// TIA Portal V19 export
FUNCTION_BLOCK "LineStates"   // FB8, LAD
{ S7_Optimized_Access := 'TRUE' }
// stored: MemoryReserve 100, SetENOAutomatically false
   VAR
      StateM1LineRunning { S7_SetPoint := 'True'} : "GenericState";
      StateM2LineRunning { S7_SetPoint := 'True'} : "GenericState";
      StateM1CurrentOrderNo { S7_SetPoint := 'True'} : "GenericState";
      StateM2CurrentOrderNo { S7_SetPoint := 'True'} : "GenericState";
      PubJsonMqttInstM1LineRunning { S7_SetPoint := 'True'} : "PublishJsonMqtt";
      PubJsonMqttInstM2LineRunning { S7_SetPoint := 'True'} : "PublishJsonMqtt";
      PubJsonMqttInstM1CurrentOrderNo { S7_SetPoint := 'True'} : "PublishJsonMqtt";
      PubJsonMqttInstM2CurrentOrderNo { S7_SetPoint := 'True'} : "PublishJsonMqtt";
      tpGen01 { S7_SetPoint := 'True'} : TP_TIME;
      tpGen02 { S7_SetPoint := 'True'} : TP_TIME;
   END_VAR
   VAR_TEMP   // added for the SCL form of the ladder/FBD networks
      _w1 : Bool;
   END_VAR
BEGIN

REGION Network 1 (SCL): Generator for data publish
   #tpGen01(IN:=NOT #tpGen02.Q,
            PT:=T#4S);

   #tpGen02(IN:=NOT #tpGen01.Q,
            PT:=T#100MS);
END_REGION

REGION Network 2: Line 1 / Machine 1 / State 'LineRunning'
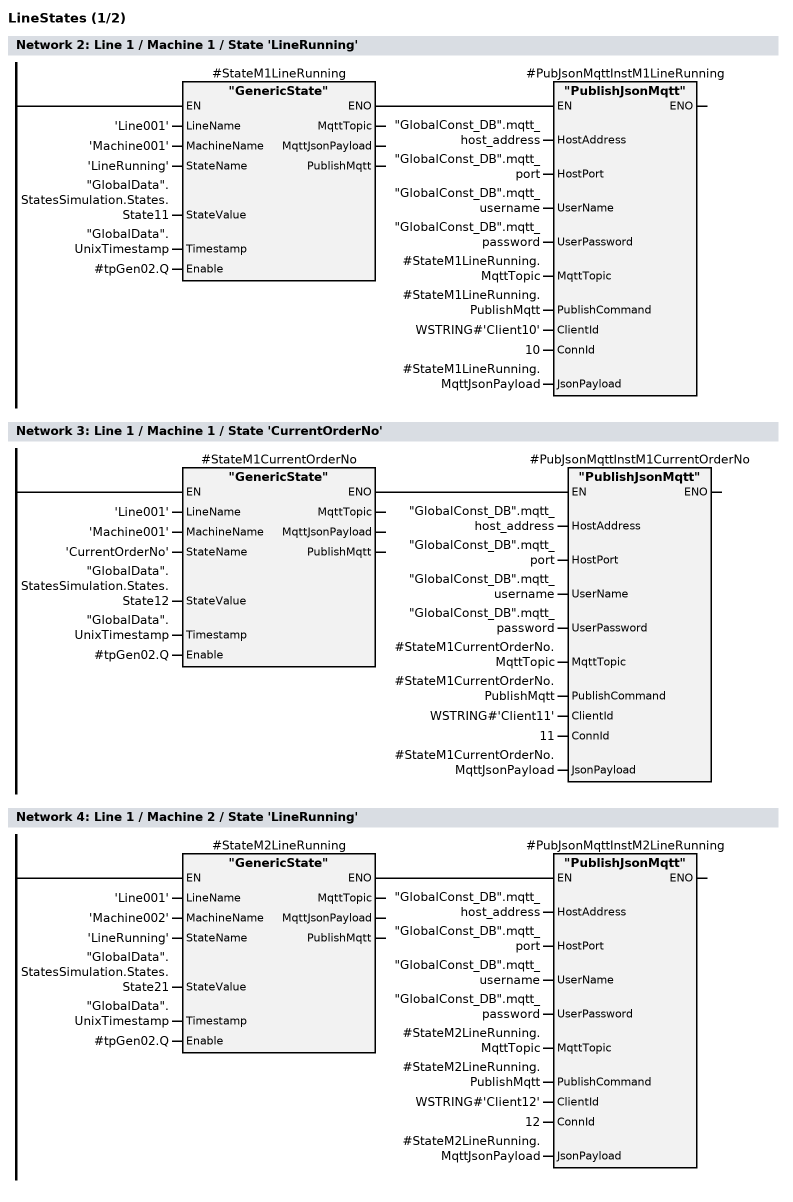
   RUNG wire#powerrail
      #StateM1LineRunning(LineName := 'Line001', MachineName := 'Machine001', StateName := 'LineRunning', StateValue := "GlobalData".StatesSimulation.States.State11, Timestamp := "GlobalData".UnixTimestamp, Enable := #tpGen02.Q, MqttTopic =>, MqttJsonPayload =>, PublishMqtt =>)
      #PubJsonMqttInstM1LineRunning(HostAddress := "GlobalConst_DB".mqtt_host_address, HostPort := "GlobalConst_DB".mqtt_port, UserName := "GlobalConst_DB".mqtt_username, UserPassword := "GlobalConst_DB".mqtt_password, MqttTopic := #StateM1LineRunning.MqttTopic, PublishCommand := #StateM1LineRunning.PublishMqtt, ClientId := WSTRING#'Client10', ConnId := 10, JsonPayload := #StateM1LineRunning.MqttJsonPayload)
   END_RUNG
   // the same network as SCL:
   #StateM1LineRunning(LineName := 'Line001',   // "GenericState"
                       MachineName := 'Machine001',
                       StateName := 'LineRunning',
                       StateValue := "GlobalData".StatesSimulation.States.State11,
                       Timestamp := "GlobalData".UnixTimestamp,
                       Enable := #tpGen02.Q,
                       ENO => #_w1);
   IF #_w1 THEN
       #PubJsonMqttInstM1LineRunning(HostAddress := "GlobalConst_DB".mqtt_host_address,   // "PublishJsonMqtt"
                               HostPort := "GlobalConst_DB".mqtt_port,
                               UserName := "GlobalConst_DB".mqtt_username,
                               UserPassword := "GlobalConst_DB".mqtt_password,
                               MqttTopic := #StateM1LineRunning.MqttTopic,
                               PublishCommand := #StateM1LineRunning.PublishMqtt,
                               ClientId := WSTRING#'Client10',
                               ConnId := 10,
                               JsonPayload := #StateM1LineRunning.MqttJsonPayload);
   END_IF;
END_REGION

REGION Network 3: Line 1 / Machine 1 / State 'CurrentOrderNo'
   RUNG wire#powerrail
      #StateM1CurrentOrderNo(LineName := 'Line001', MachineName := 'Machine001', StateName := 'CurrentOrderNo', StateValue := "GlobalData".StatesSimulation.States.State12, Timestamp := "GlobalData".UnixTimestamp, Enable := #tpGen02.Q, MqttTopic =>, MqttJsonPayload =>, PublishMqtt =>)
      #PubJsonMqttInstM1CurrentOrderNo(HostAddress := "GlobalConst_DB".mqtt_host_address, HostPort := "GlobalConst_DB".mqtt_port, UserName := "GlobalConst_DB".mqtt_username, UserPassword := "GlobalConst_DB".mqtt_password, MqttTopic := #StateM1CurrentOrderNo.MqttTopic, PublishCommand := #StateM1CurrentOrderNo.PublishMqtt, ClientId := WSTRING#'Client11', ConnId := 11, JsonPayload := #StateM1CurrentOrderNo.MqttJsonPayload)
   END_RUNG
   // the same network as SCL:
   #StateM1CurrentOrderNo(LineName := 'Line001',   // "GenericState"
                          MachineName := 'Machine001',
                          StateName := 'CurrentOrderNo',
                          StateValue := "GlobalData".StatesSimulation.States.State12,
                          Timestamp := "GlobalData".UnixTimestamp,
                          Enable := #tpGen02.Q,
                          ENO => #_w1);
   IF #_w1 THEN
       #PubJsonMqttInstM1CurrentOrderNo(HostAddress := "GlobalConst_DB".mqtt_host_address,   // "PublishJsonMqtt"
                               HostPort := "GlobalConst_DB".mqtt_port,
                               UserName := "GlobalConst_DB".mqtt_username,
                               UserPassword := "GlobalConst_DB".mqtt_password,
                               MqttTopic := #StateM1CurrentOrderNo.MqttTopic,
                               PublishCommand := #StateM1CurrentOrderNo.PublishMqtt,
                               ClientId := WSTRING#'Client11',
                               ConnId := 11,
                               JsonPayload := #StateM1CurrentOrderNo.MqttJsonPayload);
   END_IF;
END_REGION

REGION Network 4: Line 1 / Machine 2 / State 'LineRunning'
   RUNG wire#powerrail
      #StateM2LineRunning(LineName := 'Line001', MachineName := 'Machine002', StateName := 'LineRunning', StateValue := "GlobalData".StatesSimulation.States.State21, Timestamp := "GlobalData".UnixTimestamp, Enable := #tpGen02.Q, MqttTopic =>, MqttJsonPayload =>, PublishMqtt =>)
      #PubJsonMqttInstM2LineRunning(HostAddress := "GlobalConst_DB".mqtt_host_address, HostPort := "GlobalConst_DB".mqtt_port, UserName := "GlobalConst_DB".mqtt_username, UserPassword := "GlobalConst_DB".mqtt_password, MqttTopic := #StateM2LineRunning.MqttTopic, PublishCommand := #StateM2LineRunning.PublishMqtt, ClientId := WSTRING#'Client12', ConnId := 12, JsonPayload := #StateM2LineRunning.MqttJsonPayload)
   END_RUNG
   // the same network as SCL:
   #StateM2LineRunning(LineName := 'Line001',   // "GenericState"
                       MachineName := 'Machine002',
                       StateName := 'LineRunning',
                       StateValue := "GlobalData".StatesSimulation.States.State21,
                       Timestamp := "GlobalData".UnixTimestamp,
                       Enable := #tpGen02.Q,
                       ENO => #_w1);
   IF #_w1 THEN
       #PubJsonMqttInstM2LineRunning(HostAddress := "GlobalConst_DB".mqtt_host_address,   // "PublishJsonMqtt"
                               HostPort := "GlobalConst_DB".mqtt_port,
                               UserName := "GlobalConst_DB".mqtt_username,
                               UserPassword := "GlobalConst_DB".mqtt_password,
                               MqttTopic := #StateM2LineRunning.MqttTopic,
                               PublishCommand := #StateM2LineRunning.PublishMqtt,
                               ClientId := WSTRING#'Client12',
                               ConnId := 12,
                               JsonPayload := #StateM2LineRunning.MqttJsonPayload);
   END_IF;
END_REGION

REGION Network 5: Line 1 / Machine 2 / State 'CurrentOrderNo'
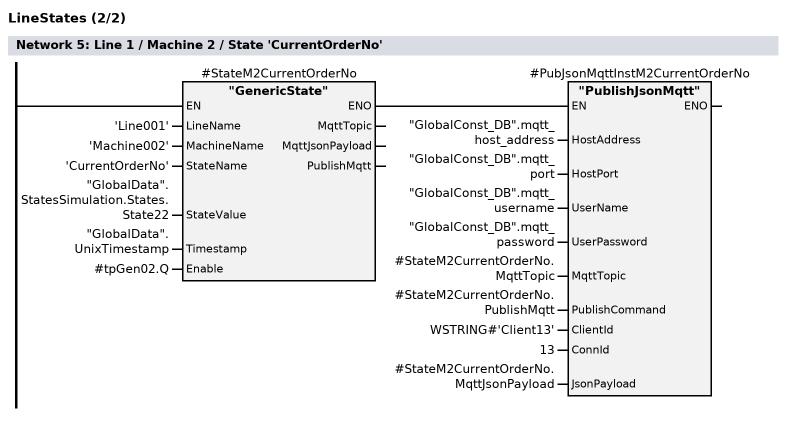
   RUNG wire#powerrail
      #StateM2CurrentOrderNo(LineName := 'Line001', MachineName := 'Machine002', StateName := 'CurrentOrderNo', StateValue := "GlobalData".StatesSimulation.States.State22, Timestamp := "GlobalData".UnixTimestamp, Enable := #tpGen02.Q, MqttTopic =>, MqttJsonPayload =>, PublishMqtt =>)
      #PubJsonMqttInstM2CurrentOrderNo(HostAddress := "GlobalConst_DB".mqtt_host_address, HostPort := "GlobalConst_DB".mqtt_port, UserName := "GlobalConst_DB".mqtt_username, UserPassword := "GlobalConst_DB".mqtt_password, MqttTopic := #StateM2CurrentOrderNo.MqttTopic, PublishCommand := #StateM2CurrentOrderNo.PublishMqtt, ClientId := WSTRING#'Client13', ConnId := 13, JsonPayload := #StateM2CurrentOrderNo.MqttJsonPayload)
   END_RUNG
   // the same network as SCL:
   #StateM2CurrentOrderNo(LineName := 'Line001',   // "GenericState"
                          MachineName := 'Machine002',
                          StateName := 'CurrentOrderNo',
                          StateValue := "GlobalData".StatesSimulation.States.State22,
                          Timestamp := "GlobalData".UnixTimestamp,
                          Enable := #tpGen02.Q,
                          ENO => #_w1);
   IF #_w1 THEN
       #PubJsonMqttInstM2CurrentOrderNo(HostAddress := "GlobalConst_DB".mqtt_host_address,   // "PublishJsonMqtt"
                               HostPort := "GlobalConst_DB".mqtt_port,
                               UserName := "GlobalConst_DB".mqtt_username,
                               UserPassword := "GlobalConst_DB".mqtt_password,
                               MqttTopic := #StateM2CurrentOrderNo.MqttTopic,
                               PublishCommand := #StateM2CurrentOrderNo.PublishMqtt,
                               ClientId := WSTRING#'Client13',
                               ConnId := 13,
                               JsonPayload := #StateM2CurrentOrderNo.MqttJsonPayload);
   END_IF;
END_REGION
END_FUNCTION_BLOCK
